FUNCTION_BLOCK FB_WorkerDefGrid_Print_WEU EXTENDS FB_WorkerDefGrid IMPLEMENTS I_PrintSubsystem
VAR_INPUT
  nPrintPos             : DINT;   // Absolute printing position [SubPx]
  fMasterSpeed          : LREAL;  // Current Speed [m/s]
  bHardwareSync         : BOOL;   // hw sync signal (chenerates a triger internally)
  bHardwareHold         : BOOL;   // hw hold signal (and fast print stop request)
  bFastStopRequest      : BOOL;   // Fast stop print request
  bPrintStopRequest     : BOOL;   // Normal synchronized print stop
  fPrintStartOffset     : LREAL;  // [m] X-Shift - StartOffset from CT Detection X0 to Print (configurative PU/PM/PG/PA ADS offset + DetectToPrintDist) [m]
  fPrintYOffset         : LREAL;  // [m] Y-Shift
  nPhDepth              : UDINT;  // [px] ph depth
  // correction live parameter
  fPUElevation          : LREAL;  // PU distance from substrate [m]
END_VAR
VAR_OUTPUT
  bPrintActive          : BOOL;   // A print is activated / started
END_VAR
VAR
  // print
  // - references
  _pAdsPg            : POINTER TO FB_ADS_PG;      // pg ads reference (for pa)
  _pAdsCam           : POINTER TO ST_ADS_CAMERA;  // camera interface PUC

  // - instances
  fbPs               : FB_PS_NewJetmap;
  fbPa               : FB_PA;
  fB_PcAdapter       : FB_PC_Adapter;
  
  // grid specific
  // - references
  _iParamMediator    : I_ParamMediator;
  // - settings
  sDefGridSettings   : ST_DefGridSettings; 

  // print corrections
  nPointCorrections  : UDINT;     // number of registered point correction handler
  iPointCorrections  : ARRAY[1..nC_NUM_POINTCORRECTIONS] OF I_GridPointCorrection;  // point corrections
  
  // - Time of flight correction of droplets
  fbDropSpeedComp    : FB_DropSpeedComp;
  bShowDropSpeedSetup : BOOL;

  // settings or helper (global or last attached ct)
  _bWorkerPrintEnable: BOOL;    // print on worker enabled 
  _nPosX0            : DINT;    // X0 for last attached CT (detected postion)
  _nPosXS            : DINT;    // XS for last attached CT (shifted print start position)
  _nPosXDelta        : DINT;    // Shift value X0 -> XS
  _fPosY             : LREAL;   // Y shift for last attached CT
  _fCurrentImgDepth  : LREAL;   // Job: current image length [m]
  _bEndless          : BOOL;    // Job: endless
  _bPaStarted        : BOOL;
  _bPaStartRequested : BOOL;
  _bPaStopping       : BOOL;
  _sJobDef           : BOOL;
  PaStartTimeout     : TON;
  rTrigHwSync        : R_TRIG;
  bBuffStopBit : BOOL;
  _bForceDefGridOff  : BOOL;    // force deformation grid stream to ph off (send 0)
  _bForceGlobalYShift: BOOL;
  _fGlobal_YShift_px : LREAL;
  _fGlobal_YShift    : LREAL;   // [m] global y- shift (special mode if no correction is active)
  
  // grid settings
  _iPhGrid           : I_Correction_Grid;
  _sPhGridHwCfg      : ST_GridHwCfg;
  // grid limit
  _fLimitCorrectionX : LREAL;     // correction limit in y (abs) [px]
  _fLimitCorrectionY : LREAL;     // correction limit in y (abs) [px]
  _bGridWasLimited : BOOL;        // streamed grid was limited
    
  // Messaging
  (*we could implement a message handler for ST_ADS_PG message interface*)

  // History
  sRepeatHistory : ARRAY[0..nC_HistorySize-1] OF ST_RepeatHistory;
  nRepeatCt : UDINT;

  // testing
  bEnVerbose : BOOL;
END_VAR
VAR PERSISTENT
  _fColumnsToPrecharge : LREAL := nC_COLUMNS_TO_PRECHARGE;
  _fStartShiftOffset   : LREAL := fC_START_SHIFT_OFFSET;
  _fStartShiftFactor   : LREAL := fC_START_SHIFT_FACTOR;
END_VAR
VAR CONSTANT
  iC_NUM_MSG               : UDINT := 5;
  nC_COLUMNS_TO_PRECHARGE  : LREAL := 2.1;
  fC_GRIDPOINT_STREAM_TIME : LREAL := 0.0025;    // time to stream one point [s]
  fC_START_SHIFT_FACTOR    : LREAL := -0.031;   //-2.4E-2;
  fC_START_SHIFT_OFFSET    : LREAL := -0.01;    //-1.0E-2;
  nC_NUM_POINTCORRECTIONS  : UDINT := 5;
  nC_HistorySize           : UDINT := 30;
END_VAR

(*
DOC:
What will be different to FB_WorkerDefGrid_Print of DMAX
- Re-Sync StartPosDetect interface with optional camera data (y-shift)
  Clear with Attach(), security clearance
- (maybe not needed) Stream grid faster to PC (we have no break for switching the CT in endless)
- New PDI StartPostion update (+print start only for first CT) --> send to NIOS or hw buffer
- PDI GridPoint stream
- New PDI PrintingLength update (after last streamed point)
- Other rules for Worker position calculation
*)

PROPERTY aPaState : STRING
GET
aPaState := fbPa.aPaState;
END_GET
END_PROPERTY

METHOD PROTECTED  Attach : BOOL
VAR_INPUT
  iCT              : I_CT;                         (*container at triggered event position*)
END_VAR
VAR
  i : UDINT;
  bCheckErr : BOOL;
  bDeformErr : BOOL;
  eDeformStep : E_DeformationStep;
END_VAR
Attach:=FALSE;

IF NOT SUPER^.Attach(iCT:=iCT) THEN
  RETURN;
END_IF

// Additional worker checks
IF _pNewAttached = 0 THEN RETURN; END_IF

// - Additional worker checks
bDeformErr := _pNewAttached^.getDeformationStatus(eDStep=>eDeformStep);   // get latest status 

  // - job is valid?
IF _pNewAttached^.pJob = 0 OR NOT _bJobActive THEN
  LogLvl(Lvl:=E_LogSeverity.Debug, Msg:='Release: no job active');
  Release(iCT:=iCT);
  RETURN;   // do not print

// CT valid & CT present
ELSIF NOT _pNewAttached^.bValid OR NOT _pNewAttached^.bProductPresent THEN
  LogLvl(Lvl:=E_LogSeverity.Debug, Msg:='Release: no produt or not valid');
  Release(iCT:=iCT);
  RETURN;   // do not print

// Ignore start due to hardware hold  
ELSIF bHardwareHold THEN
  _pNewAttached^.AbortDeformation(sReason:=EC_Print.ecPaAbortHold.Desc, Src:=_pEcSrc^, bHideLog:=TRUE);
  Release(iCT:=iCT);
  RETURN;   // do not print

// ignore new start when stop is requested
ELSIF bPrintStopRequest OR bFastStopRequest THEN
  LogLvl(Lvl:=E_LogSeverity.Debug, Msg:='Release: stop requested');
  Release(iCT:=iCT);
  RETURN;   // do not print

// - deformation started? and no deformation error so far
ELSIF bDeformErr OR eDeformStep < E_DeformationStep.cameraStarted THEN
  Release(iCT:=iCT);  // nothing to do anymore
  
// - OK attach
ELSE
  Attach := TRUE;
END_IF


// ------------------
// NOTE: we have multi-attach, take care with editing Worker globals! 


// Prepare and Start print ---------------
// - Grid udpate settings (set in WorkerDeformation during JobStart)
sDefGridSettings := _iParamMediator.sDeformationGridSettings; 

// - clear handling data 
//    done in SUPER.Attach()  push

// - Calc print positions
//  > X Position ---
_nPosX0 := _pNewAttached^.nPosPrint_X0;         // X0 "print" position for CT (should be updated to the local position domain, not the one of CTM)
_nPosXDelta :=   F_MeterToSubPixel(fPrintStartOffset, _fPrintResolution*_fSubPxResolution)                      // + PU/PM/PG shifts
               - F_MeterToSubPixel(fbDropSpeedComp.fDropPlacementError, _fPrintResolution*_fSubPxResolution);   // - drop compensation 
_nPosXS := _nPosX0 + _nPosXDelta;   // XS effective print start position
//  > Y Position ---
//   y position (with or whithout applied global y shift from correction grid)

IF _bForceDefGridOff AND _bForceGlobalYShift THEN   // special mode to force deformation grid stream off and use "mean" y-Correction as Y-shift     
  _fGlobal_YShift_px := _pNewAttached^.fDyShift;
  _fGlobal_YShift := _fGlobal_YShift_px / _fPrintResolution * 0.0254;   // px -> m
ELSE
  _fGlobal_YShift := 0;
END_IF
_fPosY :=   F_MeterToSubPixel(fPosMeter:=fPrintYOffset, fResoSubPx:=_fPrintResolution) + _fGlobal_YShift;

// error checks on position
bCheckErr := checkPrintposTiming(nStartPos:=_nPosXS, nCurrentPos:=nPrintPos);
bCheckErr := checkGridTiming(nPosXS:=_nPosXS, nPosNow:=nPrintPos);

// - Globals
fB_PcAdapter.setPrintStartPos(nX0:=_nPosXS);
fB_PcAdapter.setPrintYShift(nYShift:=FC_LREAL_TO_DINT(_fPosY));
// - Per PS (PHs)
fbPs.bPrintEnable := iCT.bValid AND iCT.bProductPresent;              // ps enables
fbPs.setGrid(sGrid:=sDefGridSettings);                                // apply correction grid settings
fbPs.setupObject(                                                     // setup print data object
  nObjId:=TO_UDINT(iCT.pCT^.iId),               // (NOTE: must be a unique id per production)
  nCopy:=1,                                     // 
  bStop:=bBuffStopBit,                          // stop after printed this object
  bDir:=FALSE, 
  nPrintStartPos:=_nPosXS,                      // 
  nImageSelection:=iCT.pCT^.sData.lPage,        // 
  nShiftedStartX:=0                             // function not used in this project
);

_pNewAttachedHdlData^.nXS := _nPosXS;           // save start pos to handling data (for calc stop pos if needed)

// Start print (initial prep->start or just start next object)
IF NOT fbPa.printStart() THEN
  LogError(Msg:='PA not ready to start at attach');
  Release(iCT := iCT);
ELSE
  // start / Update ok
  IF NOT _bPaStarted THEN 
    _bPaStartRequested := TRUE;
  END_IF
  Attach:=TRUE;
END_IF

// debug log
LogLvl(Lvl:=E_LogSeverity.Debug, F_Concat4('printStart: at XS:', TO_STRING(_nPosXS), ' ', _pNewAttached^.print(0)));  // print container
LogLvl(Lvl:=E_LogSeverity.Debug, F_Concat4(
                                      F_Concat3('> XS = X0(', TO_STRING(iCT.GetPosX0(iTracker:=_iCTTracker)), ')'),
                                      '',
                                      F_Concat3(' + shStartOffs(', TO_STRING(F_MeterToSubPixel(fPrintStartOffset, _fPrintResolution*_fSubPxResolution)), ')'),
                                      F_Concat3(' - shDropComp(', TO_STRING(F_MeterToSubPixel(fbDropSpeedComp.fDropPlacementError, _fPrintResolution*_fSubPxResolution)), ')')
                                   ));

// debug history
FOR i:=0 TO nC_HistorySize-1 DO sRepeatHistory[i].bSelected := FALSE; END_FOR   // clear selection
nRepeatCt := (nRepeatCt + 1) MOD nC_HistorySize;
sRepeatHistory[nRepeatCt].bSelected      := TRUE;
sRepeatHistory[nRepeatCt].nX0            := _nPosXS;
sRepeatHistory[nRepeatCt].fLen           := _pNewAttached^.pJob^.fImageDepth;  // + PrePost?
sRepeatHistory[nRepeatCt].fLenEffective  := _nPosXS - sRepeatHistory[SEL(nRepeatCt=0, nRepeatCt-1, nC_HistorySize-1)].nX0;
END_METHOD

PROPERTY bForceNoCorrectionButShiftMode : BOOL
SET
// special mode for LabelExpo  
// (disable deformation but use y-shift from deformation (mean) and send it via CB global y-Shift.
IF bForceNoCorrectionButShiftMode THEN
  _bForceDefGridOff := TRUE;
  _bForceGlobalYShift := TRUE;
ELSE
  _bForceDefGridOff := FALSE;
  _bForceGlobalYShift := FALSE;
END_IF
END_SET
END_PROPERTY

PROPERTY bGridWasLimited : BOOL
GET
bGridWasLimited := _bGridWasLimited;
END_GET
END_PROPERTY

PROPERTY bJobActive : BOOL
GET
bJobActive := _bJobActive;
END_GET
END_PROPERTY

PROPERTY bPausePrintCanEx : BOOL
GET
bPausePrintCanEx := FALSE; //Not implemented
END_GET
END_PROPERTY

PROPERTY bPcEnabled : BOOL
GET
bPcEnabled := fB_PcAdapter.bPcEnable;
END_GET
END_PROPERTY

PROPERTY bPrintEnabled : BOOL
GET
bPrintEnabled := _bEnable;
END_GET
END_PROPERTY

PROPERTY bPrinting : BOOL
GET
bPrinting := fbPa.bPrinting;
END_GET
END_PROPERTY

PROPERTY bPrintReady : BOOL
GET
bPrintReady := fbPa.bReady;
END_GET
END_PROPERTY

PROPERTY bQueueEmpty : BOOL
GET
bQueueEmpty := NOT fB_PcAdapter.bJobValid;
END_GET
END_PROPERTY

PROPERTY bStartPrintCanEx : BOOL
GET
bStartPrintCanEx := fbPa.bStartCanEx;
END_GET
END_PROPERTY

PROPERTY bStopPrintCanEx : BOOL
GET
bStopPrintCanEx := fbPa.bStopCanEx;
END_GET
END_PROPERTY

{attribute 'monitoring':='call'}
PROPERTY bWorkerEnable : BOOL
GET
bWorkerEnable := SUPER^.bWorkerEnable;
END_GET
SET
IF _pAdsPg = 0 THEN
  SUPER^.bWorkerEnable := bWorkerEnable;
ELSE
  // mask worker enable with group enable
  SUPER^.bWorkerEnable := bWorkerEnable AND _pAdsPg^.bEnable;  
END_IF
END_SET
END_PROPERTY

{attribute 'monitoring':='call'}
PROPERTY bWorkerPrintEnable : BOOL
GET
bWorkerPrintEnable := _bWorkerPrintEnable;
END_GET
SET
_bWorkerPrintEnable := bWorkerPrintEnable;
END_SET
END_PROPERTY

(*
  Check timing for grid stream. 
  Reports an error if grid stream is too slow (machine running too fast for streaming the grid points over PDI)
  :returns: TRUE on error
*)
METHOD PRIVATE checkGridTiming : BOOL
VAR_INPUT
  nPosXS : DINT;
  nPosNow : DINT;
END_VAR
// check for timing problems
IF fMasterSpeed <> 0 THEN

  // - check pre-charge at beginning
  IF _fColumnsToPrecharge * fC_GRIDPOINT_STREAM_TIME * _sPhGridHwCfg.nGridRoiRows >= F_SubPixelToMeter(lPosSubPx:=SEL(nPosXS-nPosNow>0, 0, nPosXS-nPosNow), fResSubPx:=_fPrintResolution*_fSubPxResolution) / fMasterSpeed  THEN
    checkGridTiming := TRUE;
    LogError('Machine too fast for grid stream (for pre-charge at attach)');
  END_IF
  
  // - check charge time needed per columns vs machine speed and grid-sizeY
  IF fC_GRIDPOINT_STREAM_TIME * _sPhGridHwCfg.nGridRoiRows >= F_SubPixelToMeter(lPosSubPx:=TO_DINT(sDefGridSettings.nGridPitchX), fResSubPx:=_fPrintResolution) / fMasterSpeed THEN
    checkGridTiming := TRUE;
    LogError('Machine too fast for grid stream (time rows per column)');
  END_IF

END_IF
END_METHOD

(*
  Check if intended print position is valid. 
  - Reports an error if print start position is not in the future
  :returns: TRUE on error
*)
METHOD checkPrintposTiming : BOOL
VAR_INPUT
  nStartPos   : DINT;   // intended start position
  nCurrentPos : DINT;   // current position
END_VAR
IF (nStartPos - nCurrentPos) < 0 THEN 
  checkPrintposTiming := TRUE;
  LogWarning(Msg:=F_Concat4('Print start position:', TO_STRING(nStartPos) ,' < Encoder position:', TO_STRING(nCurrentPos)));
END_IF
END_METHOD

// apply other corrections to camera correction/deformation
METHOD PRIVATE correctionApply : BOOL
VAR_INPUT
  pPoint : POINTER TO ST_DeformationPointAccurate;
END_VAR
VAR
  i : UDINT;
END_VAR

// here apply all PU specific corrections
// - mechanical stretch based on temperature extension (if not done in Camera)
// - banana correction
// - Y-shifts of PU
// - trapzedoial correction
// - ...


// PU Deformation correction
IF GVL_Deformation.bC_UsePUDeformation THEN
  FOR i:=1 TO nPointCorrections DO
    iPointCorrections[i].updateCorrection(pPoint:=pPoint);
  END_FOR
END_IF
END_METHOD

(*
  Limit correction to boundaries
  :return: TRUE if limited
*)
METHOD PRIVATE correctionLimit : BOOL
VAR_INPUT
  pPoint : POINTER TO ST_DeformationPointAccurate;
  pCT    : POINTER TO FB_ContainerDefGrid;
END_VAR
VAR
  bLimited : BOOL;
  nExeedX, nExeedY : LREAL;
END_VAR
// limit point correction to boundaries and inform
IF pPoint^.dx >= _fLimitCorrectionX    THEN nExeedX := pPoint^.dx; pPoint^.dx := _fLimitCorrectionX;    bLimited:=TRUE; END_IF
IF pPoint^.dx <= -1*_fLimitCorrectionX THEN nExeedX := pPoint^.dx; pPoint^.dx := -1*_fLimitCorrectionX; bLimited:=TRUE; END_IF
IF pPoint^.dy >= _fLimitCorrectionY    THEN nExeedY := pPoint^.dy; pPoint^.dy := _fLimitCorrectionY;    bLimited:=TRUE; END_IF
IF pPoint^.dy <= -1*_fLimitCorrectionY THEN nExeedY := pPoint^.dy; pPoint^.dy := -1*_fLimitCorrectionY; bLimited:=TRUE; END_IF

IF bLimited THEN
  LogLvl(Lvl:=E_LogSeverity.Debug, Msg:=F_Concat4( F_concat2('Correction limited - Point=',TO_STRING(pPoint^.index)),
                                                     F_Concat5(' (c:',TO_STRING(pPoint^.col),'/r:',TO_STRING(pPoint^.row), ') '),
                                                     F_Concat4('dx:', TO_STRING(nExeedX), 'px dy:', TO_STRING(nExeedY)),
                                                     F_Concat4('px dx_max=+/-', TO_STRING(_fLimitCorrectionX), ' dy_max=+/-', TO_STRING(_fLimitCorrectionY))
                                                  ));
END_IF

_bGridWasLimited := SEL(bLimited, FALSE, TRUE);
correctionLimit := bLimited;
END_METHOD

// current job image length in [m]
PROPERTY fImageLength : LREAL
GET
fImageLength := _fCurrentImgDepth;
END_GET
END_PROPERTY

PROPERTY fMaxPrintSpeed : LREAL
GET
fMaxPrintSpeed := 0;  // TODO: when i_pc_adapter has the info from pc/ph
END_GET
END_PROPERTY

(*
  Max. supported speed [m/s], 0 if not available
*)
{attribute 'monitoring':='call'}
PROPERTY fMaxSpeed : LREAL
GET
VAR
  nSpeedMpMin : DINT;
END_VAR
nSpeedMpMin := SEL(bWorkerEnable AND _pAdsPg <> 0, 0, _pAdsPg^.lMaxPrintSpeed);
fMaxSpeed := TO_LREAL(nSpeedMpMin)/60;
END_GET
END_PROPERTY

{attribute 'monitoring':='call'}
PROPERTY fStartShiftFactor : LREAL
GET
fStartShiftFactor := _fStartShiftFactor;
END_GET
SET
_fStartShiftFactor := fStartShiftFactor;
END_SET
END_PROPERTY

{attribute 'monitoring':='call'}
PROPERTY fStartShiftOffset : LREAL
GET
fStartShiftOffset := _fStartShiftOffset;
END_GET
SET
_fStartShiftOffset := fStartShiftOffset;
END_SET
END_PROPERTY

METHOD PROTECTED gridUpdate : BOOL
VAR_INPUT
  bEnableDeformation : BOOL;      // enable correction update, else correction (0/0) is written
  pCT : POINTER TO FB_ContainerDefGrid;
  pCTHdlData : POINTER TO ST_WorkerDefGrid_CTData;
  pMaxDx : POINTER TO LREAL;
END_VAR
VAR
  bOK : BOOL;
  fCurrentColumnPos  : LREAL; // Currently column position (of current ct)
END_VAR


//TODO: rewrite this method to look cleaner (less if else)
IF sDefGridSettings.nGridSizeX  = 0 THEN RETURN; END_IF          // avoid endless loops
IF sDefGridSettings.nGridSizeY  = 0 THEN RETURN; END_IF
IF sDefGridSettings.nGridPitchX = 0 THEN RETURN; END_IF
IF pCT = 0 THEN RETURN; END_IF
IF pCTHdlData = 0 THEN RETURN; END_IF

gridUpdate:=TRUE;

// calculate grid column position
fCurrentColumnPos := pCTHdlData^.fPosRelToAttach / (sDefGridSettings.nGridPitchX * _fSubPxResolution);   // calc grid column position relative to worker

// Check for next correction update
bOK := TRUE;
IF pCTHdlData^.nChargedCols <= sDefGridSettings.nGridSizeX THEN
  IF bEnableDeformation THEN 
    // sync deformation points
    bOK := streamCorrection(pCT:=pCT,
                            fColPos := fCurrentColumnPos, 
                            pChargedCols:=ADR(pCTHdlData^.nChargedCols), 
                            pMaxDx:=pMaxDx,
                            nAvailPoints:=pCT^.nAvailableGridPoints);
  ELSE
    // sync empty deformation points (with NO correction)
    bOK := streamNoCorrection(pChargedCols:=ADR(pCTHdlData^.nChargedCols));
  END_IF
  
END_IF

gridUpdate := bOK;
END_METHOD

METHOD InitWorkerPrint : BOOL
VAR_INPUT
  pAdsPg                : POINTER TO FB_ADS_PG;       // pg ads reference (worker prints ads)
  iDefGridParamMediator : I_ParamMediator;            // for deformation settings
  fLimitCorrectionX     : LREAL;                      // correction limit in y (abs) [px]
  fLimitCorrectionY     : LREAL;                      // correction limit in y (abs) [px]
END_VAR
IF NOT bInitialized            THEN LogError('Base Worker not initialized! call init() before'); RETURN; END_IF
IF pAdspg = 0 THEN LogError('InitWorkerPrint: invalid parameter proviced'); RETURN; END_IF
IF iDefGridParamMediator = 0   THEN bInitialized := FALSE; LogError('Invalid parameter, no valid param mediator'); RETURN; END_IF

// Worker specific init
_pAdsPg := pAdsPg;
_iParamMediator := iDefGridParamMediator;

_fLimitCorrectionX := ABS(fLimitCorrectionX);
_fLimitCorrectionY := ABS(fLimitCorrectionY);

// Print Aggregate
fbPa.bSyncAfterDone := FALSE;
fbPa.init(iPcAdapter := fB_PcAdapter, iPsInterface := fbPs);
END_METHOD

METHOD mJobPause
END_METHOD

METHOD   mJobStart
VAR_INPUT
	sJobDef	: CalmarCompPrint.I_JobDefinition;
END_VAR
// Config workers static variables
// - security release position (2 * Image Length)
_fCtSecurityReleasePos := F_MeterToSubPixel(fPosMeter:=2.1*(sJobDef.fImageDepth/1000), fResoSubPx:=_fPrintResolution*_fSubPxResolution);

IF NOT bWorkerEnable THEN RETURN; END_IF  // only if enabled

// an initial definition at jobStart/(activation)
fbPs.setupObject(nObjId:=1, nCopy:=1, bStop:=FALSE, bDir:=FALSE, nPrintStartPos:=0, nImageSelection:=0, nShiftedStartX:=0);
fbPa.jobStart(bEndless:=sJobDef.isEndless());

_fCurrentImgDepth := sJobDef.fImageDepth/1000;
_bEndless := sJobDef.isEndless();
bBuffStopBit := NOT _bEndless;

// update deformation limit by job setting
//_fLimitCorrectionX   // [px]

// grid settings update
IF _iPhGrid <> 0 THEN _sPhGridHwCfg := _iPhGrid.getGridHwCfg(); END_IF 

_bJobActive := TRUE;
END_METHOD

METHOD  mJobStop
VAR_INPUT
	sStatus	: CalmarCompPrint.I_JobStatus;
END_VAR
fbPa.jobStop();
_bJobActive := FALSE;
_bPaStarted := FALSE;
_bPaStartRequested := FALSE;
END_METHOD

METHOD mProduced
VAR_INPUT
	(* current progress*)
	sProgress	: CalmarCompPrint.I_JobProgress;
END_VAR
END_METHOD

// register additional grid correction handlers
METHOD RegisterGridCorrection : BOOL
VAR_INPUT
  iGridCorrection : I_GridPointCorrection;
END_VAR
VAR
  i : UDINT;
END_VAR
IF iGridCorrection = 0 THEN LogError('registerGridCorrection: ivalid interface, ignore'); RETURN; END_IF
IF nPointCorrections >= nC_NUM_POINTCORRECTIONS THEN LogError('registerGridCorrection: too many corrections registred, ignore'); RETURN; END_IF

nPointCorrections := nPointCorrections + 1;
iPointCorrections[nPointCorrections] := iGridCorrection;
END_METHOD

METHOD registerPc : BOOL
VAR_INPUT
  iNewPC : I_PC;
END_VAR
registerPc := fB_PcAdapter.registerPc(iNewPC := iNewPC);
END_METHOD

METHOD registerPh : BOOL
VAR_INPUT
  iPH : I_PH;
END_VAR
//Attach head to print station
IF iPH <> 0 THEN
  fbPs.registerPh(iNewPh:=iPH);
  _iPhGrid := iPH.iGridCorrection;
END_IF
END_METHOD

(*
  Release CT from Worker.
  :return: TRUE if CT was released, FALSE if no CT was registered 
*)
METHOD Release : BOOL
VAR_INPUT
  iCT              : I_CT;                         (*container at triggered event position*)
END_VAR

Release := SUPER^.Release(iCT:=iCT);
END_METHOD

// Release all attached CTs
METHOD PRIVATE ReleaseAllAttached
VAR
  i : UDINT;
  pCt : POINTER TO FB_ContainerDefGrid;
END_VAR
//Work only with attached container
IF _nAttachedCTs = 0 THEN RETURN; END_IF
  
FOR i:=nLowerIndexCTList TO nLowerIndexCTList + _nAttachedCTs - 1 DO
  pCt := _pAttachedCTList[i];
  pCt^.AbortDeformation(sReason:=EC_Print.ecPaAbortHold.Desc, Src:=_pEcSrc^, bHideLog:=TRUE);
  
  Release(iCT:=pCt^);
END_FOR
END_METHOD

METHOD PRIVATE setupPosition
VAR
  fPreStartShift : LREAL;
  fCalculatedWorkerPos : LREAL;
END_VAR
IF _pAttachedCt <> 0 THEN RETURN; END_IF   // Update only without attached container

// Worker position update
fPreStartShift := (_fStartShiftOffset + _fStartShiftFactor * fMasterSpeed);
fCalculatedWorkerPos := fPrintStartOffset + fPreStartShift;
IF _fWorkerPosition <> fCalculatedWorkerPos THEN   // Worker position changed
  fPosition := fCalculatedWorkerPos;  // Update worker position
END_IF
END_METHOD

METHOD PRIVATE sim
END_METHOD

METHOD PRIVATE streamCorrection : BOOL
VAR_INPUT
  pCT : POINTER TO FB_ContainerDefGrid;
  fColPos : LREAL;  // current column position (relative to Attach-Pos)
  pChargedCols : POINTER TO UDINT;  // number of already charged columns (pointer for internal edit)
  pMaxDx : POINTER TO LREAL;
  nAvailPoints : UDINT;     // available gridPoints on CT
END_VAR
VAR
  nRow : UDINT;
  bWasSet : BOOL;
  sPoint : ST_DeformationPointAccurate;
  fCurrentPreCharge  : LREAL; // Currently to be precharged (for scope)
END_VAR
VAR_INST
  nAvailPoints_mem : UDINT;
END_VAR
IF pChargedCols = 0 THEN RETURN; END_IF

streamCorrection := TRUE;

fCurrentPreCharge := fColPos + _fColumnsToPrecharge;

WHILE pChargedCols^ < LIMIT(0, FLOOR(fCurrentPreCharge), sDefGridSettings.nGridSizeX) DO
  
  IF nAvailPoints >= sDefGridSettings.nGridSizeY * (pChargedCols^+1) THEN     // Complete next column available?
    
    nAvailPoints_mem := 0;
    LogLvl(Lvl:=E_LogSeverity.Debug, Msg:=F_Concat4('CT: ', TO_STRING(pCT^.pCT^.iId),' Charge CG col: ', TO_STRING(pChargedCols^)));
    
    pMaxDx^ := 0;   // per columns
    
    FOR nRow := 0 TO sDefGridSettings.nGridSizeY - 1 DO
      
      // get points
      IF pCT^.getDeformationPoint(nCol:=pChargedCols^, nRow:=nRow, nSel:=0, sPoint=>sPoint, bWasSet=>bWasSet) THEN
        
        IF NOT bWasSet THEN LogWarning(F_Concat5('Point[c(',TO_STRING(pChargedCols^),')/r(', TO_STRING(nRow),')] was not set')); END_IF
        
        // apply PU corrections
        correctionApply(pPoint:=ADR(sPoint));
        
        // limitation corrections
        correctionLimit(pPoint:=ADR(sPoint), pCT:=pCt);
        
        // max. dx tracing
        IF sPoint.dx > pMaxDx^ THEN pMaxDx^ := sPoint.dx; END_IF
        
        // send point
        IF NOT fbPs.newGridPoint(sPoint:=sPoint) THEN
          // err
          LogError(Msg:='stream new point failed');
          streamCorrection:=FALSE;
          RETURN;
        ELSE
          // ok
          pCT^.storeStreamedDeformationPoint(pPoint:=ADR(sPoint));    // save to sent table
          IF bEnVerbose THEN
            F_Concat3( 
              F_concat2('Send Point=',TO_STRING(sPoint.index)),
              F_Concat5(' (c:',TO_STRING(sPoint.col),'/r:',TO_STRING(sPoint.row), ')'),
              F_Concat4(' dx=', TO_STRING(sPoint.dx), ' dy=', TO_STRING(sPoint.dy))
            );
          END_IF
        END_IF
      ELSE
        LogError(Msg:='get new grid point failed');
        streamCorrection:=FALSE;
      END_IF
    END_FOR
    
    pChargedCols^ := pChargedCols^ + 1;
  ELSE
    
    // not yet enought points for next full column
    IF nAvailPoints > nAvailPoints_mem THEN // log once or after every update of new available points
      LogLvl(Lvl:=E_LogSeverity.Error, Msg:=F_Concat3(
                                            F_Concat2('CT: ', TO_STRING(pCT^.pCT^.iId)), 
                                            F_Concat2(' Print column expected but not available. Avil=', TO_STRING(nAvailPoints)),
                                            F_Concat2(' of expected: ', TO_STRING(sDefGridSettings.nGridSizeY * (pChargedCols^+1)))
                                          ));
    END_IF
    nAvailPoints_mem := nAvailPoints;
    streamCorrection:=FALSE;
    RETURN;
  END_IF
  
END_WHILE
END_METHOD

METHOD PRIVATE streamNoCorrection : BOOL
VAR_INPUT
  pChargedCols : POINTER TO UDINT;  // number of already charged columns (pointer for internal edit)
END_VAR
VAR
  nRow : UDINT;
  sPoint : ST_DeformationPointAccurate;
END_VAR
IF pChargedCols = 0 THEN RETURN; END_IF

// send points with no deformation
FOR nRow := 0 TO sDefGridSettings.nGridSizeY - 1 DO
    MEMSET(destAddr:=ADR(sPoint), fillByte:=0, n:=SIZEOF(sPoint));
    sPoint.col := TO_DINT(pChargedCols^);
    sPoint.row := TO_DINT(nRow);
    IF NOT fbPs.newGridPoint(sPoint:=sPoint) THEN
       LogError(Msg:='stream new point failed');
       streamNoCorrection:=FALSE;
       RETURN;
    END_IF
END_FOR

// select next column
pChargedCols^ := pChargedCols^ + 1;

streamNoCorrection := TRUE;
END_METHOD

METHOD work
VAR
  bDeformErr : BOOL;
  nDeformStep : E_DeformationStep;
  i : UDINT;
  pCt : POINTER TO FB_ContainerDefGrid;
  pCtHdlData : POINTER TO ST_WorkerDefGrid_CTData;
  nUpdateStopPos : DINT;
  fMaxDx : LREAL;
END_VAR
IF _iParamMediator = 0 THEN F_Report_Error(ErrType:=EN_REPORT_ERROR_TYPE.Report_Error_0Pointer); RETURN; END_IF
bError := FALSE; nError := 0;

setupPosition();  // calculate and set worker position

SUPER^.work();

(*Print correction*)
fbDropSpeedComp(fMasterSpeed:=fMasterSpeed, fDropTravelDistance:=fPUElevation);

(*Update virtual encoder on all controller boards*)
fB_PcAdapter.setEncoderPos(nPrintPos);
fB_PcAdapter();

(*Call print aggregate*)
rTrigHwSync(CLK:=bHardwareSync); 
IF rTrigHwSync.Q THEN fbPa.sync(); END_IF   // external sync cmd

// PA control
fbPa.bHold := bHardwareHold;                // external hw hold, NOTE: this stop the current print iPC.stop()
fbPa();
PaStartTimeout(IN:=_bPaStartRequested, PT:=fbPa.fbStatePrepare.tC_PrepareTimeout+T#10MS);

IF _bPaStartRequested THEN
  // Starting...
  IF fbPa.bPrinting THEN
    // started
    _bPaStarted := TRUE; 
    _bPaStartRequested := FALSE;
  ELSIF PaStartTimeout.Q THEN     // Abort print
    // start timeout -> abort
    _bPaStarted := FALSE;
    _bPaStartRequested := FALSE;
    fbPa.printStop(bSyncedStop:=FALSE);
    ReleaseAllAttached();
  END_IF
ELSIF _bPaStarted THEN
  // - Started... Supervision of FSM
  IF fbPa.bDone OR fbPa.bStop THEN  // if pa did stop
    _bPaStarted := FALSE; 
    ReleaseAllAttached();
  (*ELSIF fbpa.bError THEN
    ReleaseAllAttached();*)
	END_IF 
  // - disabled
  IF NOT bWorkerEnable THEN
    _bPaStarted := FALSE;
    fbPa.printStop(bSyncedStop:=FALSE);
    ReleaseAllAttached();
  END_IF
  // - machine stopped
  IF bFastStopRequest OR bHardwareHold THEN
    _bPaStarted := FALSE;
    fbPa.printStop(bSyncedStop:=FALSE);
    ReleaseAllAttached();
	END_IF
  // - Synced stopping request
  IF bPrintStopRequest THEN
    IF NOT _bPaStopping THEN  _bPaStopping := TRUE;
      fbPs.stopObject(nObjId:=0, 
                      nStopPosition:=   _nPosXS           // use last used/calculated XS
                                      + F_MeterToSubPixel(fPosMeter:=_fCurrentImgDepth + 0.05, fResoSubPx:=_fPrintResolution*_fSubPxResolution)
                                      + TO_DINT(nPhDepth*_fSubPxResolution));
      fbPa.printStop(bSyncedStop:=TRUE);                  // should stop automatically when all buffer are done   
     END_IF
  ELSE
    _bPaStopping := FALSE;
  END_IF
END_IF

bPrintActive := _bPaStarted;


// for all attached CTs ----------------
// - Disable      -> PA.Stop, tag all as error, release all [OK]
// - FastStop     -> PA.Stop, tag all as error, release all [  ]
// - Hold         -> PA.Hold => PC.stop() [  ]
// - PA Starting  ->  [  ]
// - JobStop      -> PA.jobStop() -> tag all as error, release all [  ]
// - Normal Stop  -> PS.Request a stop [  ]
// - OK           =>  GridStream -> Release when all done [  ]
FOR i:=nLowerIndexCTList TO nLowerIndexCTList + _nAttachedCTs - 1 DO
  pCt := _pAttachedCTList[i];
  // Handling Data
  // - fPosRelToAttach: position relative to attach
  // - nChargedCols: charged columns
  // - nData2: not used
  // - fData1: not used
  // - fData2: not used
  pCtHdlData := ADR(_stAttachedCTData[i]);
  
  // Grid update
  bDeformErr := pCt^.getDeformationStatus(eDStep=>nDeformStep);
  IF NOT bDeformErr AND nDeformStep >= E_DeformationStep.gridStarted AND NOT _bForceDefGridOff THEN
    IF NOT gridUpdate(bEnableDeformation:=TRUE, pCT:=pCt, pCTHdlData:=pCtHdlData, pMaxDx:=ADR(fMaxDx)) THEN
      pCt^.AbortDeformation(sReason:='deformation point update failed', Src:=_pEcSrc^, bHideLog:=FALSE);
    END_IF
  ELSE
    // not started or error already --> erase deformation points and send no correction points
    IF NOT gridUpdate(bEnableDeformation:=FALSE, pCT:=pCt, pCTHdlData:=pCtHdlData, pMaxDx:=ADR(fMaxDx)) THEN
      pCt^.AbortDeformation(sReason:='deformation point update failed', Src:=_pEcSrc^, bHideLog:=FALSE);
    END_IF
  END_IF
  
  // RELEASE when Grid stream finished
  IF pCtHdlData^.nChargedCols >= sDefGridSettings.nGridSizeX THEN
    IF NOT _bEndless THEN // single print mode
      // Update print length in single print mode
      nUpdateStopPos := pCtHdlData^.nXS                                                                                   // XS print start position
                      + F_MeterToSubPixel(fPosMeter:=_fCurrentImgDepth, fResoSubPx:=_fPrintResolution*_fSubPxResolution)  // sheet length
                      + F_MeterToSubPixel(fPosMeter:=fMaxDx, fResoSubPx:=_fPrintResolution)                               // max. deformation
                      + TO_DINT(nPhDepth*_fSubPxResolution);
      fbPs.stopObject(nObjId:=0, nStopPosition:=nUpdateStopPos);        // update (overwrite firmware internal calculated) jm stop position
      LogLvl(Lvl:=E_LogSeverity.Debug, Msg:=F_Concat6('Update StopPos=', TO_STRING(nUpdateStopPos),' (',F_UDINT_TO_HEXSTR(lVal:=TO_UDINT(nUpdateStopPos), bLower:=FALSE), ') on ', pCt^.print(format:=0)));
    END_IF
    Release(pCt^);
  END_IF
END_FOR


// forward pa state to pg ads
IF _pAdsPg <> 0 THEN
  _pAdsPg^.aState := fbPa.aPaState;
  _pAdsPg^.lError := nError; 
  _pAdsPg^.bError := bError;
END_IF


// logging config
fbPa.LogLevel := LogLevel;
fB_PcAdapter.LogLevel := LogLevel;

sim();
END_METHOD

END_FUNCTION_BLOCK

(* stored: Version 1.1.0.1, ProductVersion 3.1.4024.11
   POU FB_WorkerDefGrid_Print_WEU: Id {40ec5b58-a08c-49a3-8c49-35e7e7ec45f8}, SpecialFunc None
   Folder Grid: Id {7717ddbf-7386-45fa-9de0-515fcc94e8e4}
   Folder helper: Id {f35db832-3481-4603-9394-12ac1e914d8b}
   Folder I_PrintStatusClient: Id {84a612a8-b7a1-414c-86f6-e5f652351528}
   Folder I_PrintSubsystem: Id {89eea201-cc9b-42a7-b203-b799f001e8a5}
   Property aPaState: Id {602b3711-53fa-4c45-b7c9-b07a17bff4b0}
   Get Get: Id {50e62729-2f8b-4a88-9511-d9d56e72c66e}
   Method Attach: Id {f3116540-c949-4fd3-8ec5-e9b8a0b92e19}
   Property bForceNoCorrectionButShiftMode: Id {0e805a25-53a1-4446-82ba-bdcca0a95608}
   Set Set: Id {4741b186-fe43-4db5-94de-23698d755f67}
   Property bGridWasLimited: Id {cba7a0fa-4cf6-47aa-9516-8de8a7c89812}
   Get Get: Id {4693dddc-f428-4e62-b783-d362d65e30e9}
   Property bJobActive: Id {8d05e057-9131-4682-b6e9-f206f93057fd}
   Get Get: Id {635dcf08-0a3c-4c91-b00e-013bfbbe8d62}
   Property bPausePrintCanEx: Id {c9206e32-815b-4ac5-8772-1e5e371622f0}
   Get Get: Id {468a2e22-f6e5-4928-856f-8f12e1ed7d7c}
   Property bPcEnabled: Id {f78dfe83-9c36-4589-a069-d10c1501f7d5}
   Get Get: Id {06dae430-a691-4272-850d-14968118c35b}
   Property bPrintEnabled: Id {2be79ade-9a03-49a3-8512-bf19048a6f97}
   Get Get: Id {30b42fbb-6c2c-4ca7-8e66-f6de3af95767}
   Property bPrinting: Id {35a5ef32-6a49-462c-97d4-5aab8d1d4440}
   Get Get: Id {b31847aa-fc02-4d08-96a1-1b060aa7784e}
   Property bPrintReady: Id {ed2d0eb3-4bca-4da9-9609-d463532fb456}
   Get Get: Id {a979108d-94c6-4426-b528-c70b835a487e}
   Property bQueueEmpty: Id {e5838cfc-96f0-4053-8d89-ebac33d76414}
   Get Get: Id {8e6341a9-54d0-4d40-940c-849af16f8cf8}
   Property bStartPrintCanEx: Id {c6548741-3838-48b4-94a2-2c713b449793}
   Get Get: Id {55d13fb0-65ad-4f10-adb5-b0a04d461ef4}
   Property bStopPrintCanEx: Id {8de99977-22b4-4b56-9ce7-e2715ec2c5d8}
   Get Get: Id {7449a1b2-3c6c-4fa7-8db2-34a4762eded1}
   Property bWorkerEnable: Id {a239c405-3b41-4955-afc6-bf6db6144aba}
   Get Get: Id {2994a149-d3b5-43a3-abea-57b75c0b16f3}
   Set Set: Id {4b62668b-935f-4eb5-9ea1-258551a03816}
   Property bWorkerPrintEnable: Id {e896c398-eb58-419f-a62e-e477b9eb7018}
   Get Get: Id {b0994bc0-6e24-439d-8670-f69c530efb04}
   Set Set: Id {9a3fbfdf-f14d-45da-86f6-4e2244cc0857}
   Method checkGridTiming: Id {074a2fa5-30e2-49b9-a0af-b54ac7a7046e}
   Method checkPrintposTiming: Id {4d37968d-ec12-4c9f-af77-8b90fd88ac52}
   Method correctionApply: Id {3896ed9a-7df9-4b49-b21e-0f6e5567045a}
   Method correctionLimit: Id {57d61141-2a56-438f-bc2b-30a98aedb0c5}
   Property fImageLength: Id {cf67713d-56b0-4ab7-bfef-5590483cb262}
   Get Get: Id {d7dae5b3-794e-4710-8422-40213b70827c}
   Property fMaxPrintSpeed: Id {32d1506f-ef65-413b-a0e1-e8e167a55813}
   Get Get: Id {4aa29dae-4af7-4804-8f6f-42f5c22017d7}
   Property fMaxSpeed: Id {f9f94698-f027-43f9-934a-e9b9530d8364}
   Get Get: Id {e28a9980-a7d4-4d01-8341-ad20142e00a5}
   Property fStartShiftFactor: Id {fba4b82c-d8d7-4aa8-9961-37223fc7399d}
   Get Get: Id {9583c940-e223-4593-ab6d-56ccd53d65c6}
   Set Set: Id {d8a12295-b18f-40c5-9499-a4a4a30ce248}
   Property fStartShiftOffset: Id {a4f69a23-d8af-4180-91ac-e18bbceab061}
   Get Get: Id {f28186a0-8b84-4a1d-bfdf-468140ca1a89}
   Set Set: Id {3d7e6a57-45de-429b-9d8f-195666ea6671}
   Method gridUpdate: Id {d439af6b-1409-49a3-9972-8e6454eaa4c5}
   Method InitWorkerPrint: Id {11ead43b-c38a-4634-aeeb-b2b155209088}
   Method mJobPause: Id {f3eed637-6d91-4944-b32f-62103cfbc23c}
   Method mJobStart: Id {fad66dc0-701c-4926-8431-0a890852145c}
   Method mJobStop: Id {be6a759a-0a7c-431c-a6c5-4123eab0e065}
   Method mProduced: Id {8b03a2b7-20e3-4aed-962c-7b216052cfd2}
   Method RegisterGridCorrection: Id {bd4e00d1-d0f9-4d2c-8f20-4113d76a8b41}
   Method registerPc: Id {c8e6b13d-1305-4afa-b5e0-db419018a599}
   Method registerPh: Id {fc615e5b-94b3-4925-ad1c-9fd4847922b3}
   Method Release: Id {3db161bd-cbd6-4efd-b1ba-ff0f576acda0}
   Method ReleaseAllAttached: Id {b4d3805d-206f-4b57-a74a-eac65302b829}
   Method setupPosition: Id {26647d66-6785-4cbd-9f08-bccca3128f00}
   Method sim: Id {9e7594b8-df13-406a-8276-6aa107308d4a}
   Method streamCorrection: Id {9a2284d8-c925-4f99-9d0a-d6f0de9d1180}
   Method streamNoCorrection: Id {1322f48f-faf9-4d70-b764-a60a64c0ed15}
   Method work: Id {4730ace3-b65a-4c30-b41a-687d4f7038b3} *)
